KUKA KRL data list: ChangeTool.dat

&ACCESS RV
DEFDAT ChangeTool PUBLIC

ENDDAT
